RoboDK station: milling.rdk

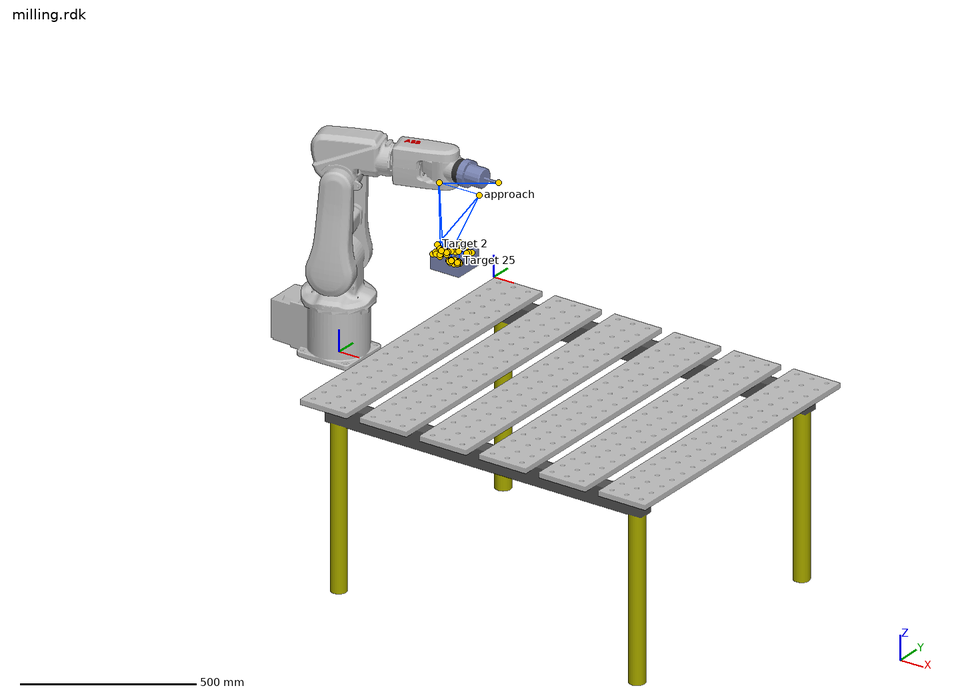
[picture v0: the station drawn from its stored meshes, robots at their saved joint values, targets as dots, program paths as lines]
Station template (saved by RoboDK 5.3.4). Poses are relative to the parent item; angles as X-Y-Z fixed-axis rotations.
  - frame ABB IRB 120-3/0.6 Base at (0, 0, 0) mm
    - robot ABB IRB 120-3/0.6: 6 axes, payload 3 kg, reach 580 mm, repeatability 0.01 mm, weight 25 kg
        modified DH rows (alpha deg, a mm, theta deg, d mm): 0, 0, 0, 290; -90, 0, -90, 0; 0, 270, 0, 0; -90, 70, 0, 302; 90, 0, 0, 0; -90, 0, 180, 72
        joint limits [-165, -110, -90, -160, -120, -400] to [165, 110, 70, 160, 120, 400]; home [0, 0, 0, 0, 0, 0]; saved at [17.579, 3.209, -3.289, -89.746, 17.579, 89.734]
      - tool AssemblyMillCutter, TCP at (0, 0, 112.79) mm, size 80 x 120 x 80 mm
  - object Table at (800, 0, 100) mm, size 1193.8 x 965.2 x 609.6 mm, geometry from welding_table.sld
  - frame worktable at (200, 480, 100) mm
    - object Task3_Part at (250, -430, 280) mm, rotated rx 90 ry 0 rz -180 deg, size 100 x 50 x 100 mm, geometry from Task3_Part.STEP
    - target approach (Cartesian target) at (287, -480, 530) mm, rotated rx 0 ry 90 rz 0 deg; joints [0, 0, 0, 0, 0, 0] of ABB IRB 120-3/0.6
    - target Target 2 (Cartesian target) at (150, -493.7, 340) mm, rotated rx -180 ry 0 rz -90 deg; joints [-2.242, 10.254, -10.083, 0, 89.83, -92.242] of ABB IRB 120-3/0.6
    - target Target 3 (Cartesian target) at (150, -493.7, 320) mm, rotated rx 180 ry 0 rz -90 deg; joints [-2.242, 9.393, -5.327, 0, 85.934, -92.242] of ABB IRB 120-3/0.6
    - target Target 4 (Cartesian target) at (176, -493.7, 320) mm, rotated rx 180 ry 0 rz -90 deg; joints [-2.087, 15.254, -12.292, 0, 87.038, -92.087] of ABB IRB 120-3/0.6
    - target Target 5 (Cartesian target) at (176, -515.9, 320) mm, rotated rx 180 ry 0 rz -90 deg; joints [-5.454, 15.592, -12.71, 0, 87.118, -95.454] of ABB IRB 120-3/0.6
    - target Target 6 (Cartesian target) at (150, -515.9, 320) mm, rotated rx 180 ry 0 rz -90.94 deg; joints [-5.856, 9.74, -5.724, 0, 85.985, -94.918] of ABB IRB 120-3/0.6
    - target Target 7 (Cartesian target) at (150, -501, 320) mm, rotated rx -180 ry 0 rz -90.94 deg; joints [-3.434, 9.473, -5.418, 0, 85.945, -92.496] of ABB IRB 120-3/0.6
    - target Target 8 (Cartesian target) at (170, -501, 320) mm, rotated rx -180 ry 0 rz -90.94 deg; joints [-3.248, 13.955, -10.703, 0, 86.748, -92.31] of ABB IRB 120-3/0.6
    - target Target 9 (Cartesian target) at (157, -508, 320) mm, rotated rx -180 ry 0 rz -90.94 deg; joints [-4.485, 11.132, -7.339, 0, 86.207, -93.547] of ABB IRB 120-3/0.6
    - target Target 10 (Cartesian target) at (170, -508, 320) mm, rotated rx -180 ry 0 rz -90.94 deg; joints [-4.328, 14.06, -10.831, 0, 86.771, -93.39] of ABB IRB 120-3/0.6
    - target Target 11 (Cartesian target) at (170, -508, 340) mm, rotated rx -180 ry 0 rz -90.94 deg; joints [-4.328, 15.03, -15.796, 0, 90.765, -93.39] of ABB IRB 120-3/0.6
    - target Target 24 (Cartesian target) at (194, -444, 340) mm, rotated rx -180 ry 0 rz -90 deg; joints [5.221, 21.03, -23.466, 0, 92.436, -84.779] of ABB IRB 120-3/0.6
    - target Target 13 (Cartesian target) at (194, -444, 320) mm, rotated rx -180 ry 0 rz -90 deg; joints [5.221, 19.845, -18.11, 0, 88.265, -84.779] of ABB IRB 120-3/0.6
    - target Target 14 (Cartesian target) at (236, -444, 320) mm, rotated rx -180 ry 0 rz -90 deg; joints [4.72, 30.95, -33.475, 0, 92.525, -85.28] of ABB IRB 120-3/0.6
    - target Target 15 (Cartesian target) at (236, -466, 320) mm, rotated rx 180 ry 0 rz -90 deg; joints [1.839, 30.578, -32.93, 0, 92.352, -88.161] of ABB IRB 120-3/0.6
    - target Target 16 (Cartesian target) at (194, -466, 320) mm, rotated rx 180 ry 0 rz -90 deg; joints [2.035, 19.507, -17.671, 0, 88.164, -87.965] of ABB IRB 120-3/0.6
    - target Target 17 (Cartesian target) at (194, -450, 320) mm, rotated rx -180 ry 0 rz -90 deg; joints [4.354, 19.724, -17.952, 0, 88.228, -85.646] of ABB IRB 120-3/0.6
    - target Target 18 (Cartesian target) at (229, -450, 320) mm, rotated rx -180 ry 0 rz -90 deg; joints [4, 28.797, -30.354, 0, 91.557, -86] of ABB IRB 120-3/0.6
    - target Target 19 (Cartesian target) at (229, -460, 320) mm, rotated rx -180 ry 0 rz -90 deg; joints [2.669, 28.633, -30.119, 0, 91.486, -87.331] of ABB IRB 120-3/0.6
    - target Target 20 (Cartesian target) at (200, -460, 320) mm, rotated rx -180 ry 0 rz -90 deg; joints [2.862, 21.036, -19.67, 0, 88.635, -87.138] of ABB IRB 120-3/0.6
    - target Target 21 (Cartesian target) at (200, -455, 320) mm, rotated rx -180 ry 0 rz -90 deg; joints [3.576, 21.105, -19.762, 0, 88.657, -86.424] of ABB IRB 120-3/0.6
    - target Target 22 (Cartesian target) at (225, -455, 320) mm, rotated rx -180 ry 0 rz -90 deg; joints [3.366, 27.593, -28.639, 0, 91.046, -86.634] of ABB IRB 120-3/0.6
    - target Target 23 (Cartesian target) at (225, -455, 340) mm, rotated rx -180 ry 0 rz -90 deg; joints [3.366, 29.282, -34.912, 0, 95.63, -86.634] of ABB IRB 120-3/0.6
    - target Target 40 (Cartesian target) at (225, -494, 340) mm, rotated rx -180 ry 0 rz -90 deg; joints [-1.887, 29.131, -34.693, 0, 95.562, -91.887] of ABB IRB 120-3/0.6
    - target Target 25 (Cartesian target) at (225, -494, 310) mm, rotated rx 180 ry 0 rz -90 deg; joints [-1.887, 26.832, -25.67, 0, 88.838, -91.887] of ABB IRB 120-3/0.6
    - target Target 26 (Cartesian target) at (235.62, -501.66, 310) mm, rotated rx -180 ry 0 rz -90 deg; joints [-2.847, 29.827, -29.932, 0, 90.105, -92.847] of ABB IRB 120-3/0.6
    - target Target 27 (Cartesian target) at (225, -516, 310) mm, rotated rx 180 ry 0 rz -90 deg; joints [-4.842, 27.177, -26.154, 0, 88.977, -94.842] of ABB IRB 120-3/0.6
    - target Target 28 (Cartesian target) at (210, -516, 310) mm, rotated rx -180 ry 0 rz -90 deg; joints [-5.018, 23.306, -20.817, 0, 87.511, -95.018] of ABB IRB 120-3/0.6
    - target Target 29 (Cartesian target) at (199.38, -508.34, 310) mm, rotated rx 180 ry 0 rz -90 deg; joints [-4.059, 20.546, -17.146, 0, 86.6, -94.059] of ABB IRB 120-3/0.6
    - target Target 30 (Cartesian target) at (210, -494, 310) mm, rotated rx 180 ry 0 rz -90 deg; joints [-1.956, 22.97, -20.365, 0, 87.394, -91.956] of ABB IRB 120-3/0.6
    - target Target 31 (Cartesian target) at (225, -494, 310) mm, rotated rx -180 ry 0 rz -90 deg; joints [-1.887, 26.832, -25.67, 0, 88.838, -91.887] of ABB IRB 120-3/0.6
    - target Target 32 (Cartesian target) at (232, -501, 310) mm, rotated rx -180 ry 0 rz -90 deg; joints [-2.783, 28.806, -28.465, 0, 89.659, -92.783] of ABB IRB 120-3/0.6
    - target Target 33 (Cartesian target) at (232, -510, 310) mm, rotated rx -180 ry 0 rz -90 deg; joints [-3.972, 28.953, -28.675, 0, 89.722, -93.972] of ABB IRB 120-3/0.6
    - target Target 34 (Cartesian target) at (204, -510, 310) mm, rotated rx -180 ry 0 rz -90 deg; joints [-4.247, 21.7, -18.667, 0, 86.967, -94.247] of ABB IRB 120-3/0.6
    - target Target 35 (Cartesian target) at (204, -500, 310) mm, rotated rx -180 ry 0 rz -90 deg; joints [-2.834, 21.548, -18.466, 0, 86.918, -92.834] of ABB IRB 120-3/0.6
    - target Target 36 (Cartesian target) at (227, -500, 310) mm, rotated rx -180 ry 0 rz -90 deg; joints [-2.682, 27.431, -26.512, 0, 89.081, -92.682] of ABB IRB 120-3/0.6
    - target Target 37 (Cartesian target) at (227, -505, 310) mm, rotated rx -180 ry 0 rz -90 deg; joints [-3.351, 27.502, -26.612, 0, 89.11, -93.351] of ABB IRB 120-3/0.6
    - target Target 38 (Cartesian target) at (207, -505, 310) mm, rotated rx -180 ry 0 rz -90 deg; joints [-3.515, 22.355, -19.54, 0, 87.185, -93.515] of ABB IRB 120-3/0.6
    - target Target 39 (Cartesian target) at (207, -505, 340) mm, rotated rx -180 ry 0 rz -90 deg; joints [-3.515, 24.197, -27.736, 0, 93.539, -93.515] of ABB IRB 120-3/0.6
    - target Target 48 (Cartesian target) at (140, -454, 305) mm, rotated rx -90 ry 0 rz -90 deg; joints [9.51, -28.081, 64.551, 15.739, -37.522, -102.6] of ABB IRB 120-3/0.6
    - target Target 41 (Cartesian target) at (160, -454, 305) mm, rotated rx -90 ry 0 rz -90 deg; joints [8.441, -22.18, 61.05, 13.304, -39.634, -100.321] of ABB IRB 120-3/0.6
    - target Target 42 (Cartesian target) at (160, -462.23, 310.75) mm, rotated rx -90 ry 0 rz -90 deg; joints [5.793, -23.239, 60.543, 9.503, -37.686, -97.546] of ABB IRB 120-3/0.6
    - target Target 43 (Cartesian target) at (160, -466, 305) mm, rotated rx -90 ry 0 rz -90 deg; joints [4.568, -22.569, 61.296, 7.279, -38.953, -95.672] of ABB IRB 120-3/0.6
    - target Target 44 (Cartesian target) at (160, -462.23, 299.55) mm, rotated rx -90 ry 0 rz -90 deg; joints [5.793, -21.695, 61.866, 8.938, -40.516, -96.818] of ABB IRB 120-3/0.6
    - target Target 45 (Cartesian target) at (160, -454, 305) mm, rotated rx -90 ry 0 rz -90 deg; joints [8.441, -22.18, 61.05, 13.304, -39.634, -100.321] of ABB IRB 120-3/0.6
    - target Target 46 (Cartesian target) at (160, -460, 305) mm, rotated rx -90 ry 0 rz -90 deg; joints [6.512, -22.403, 61.191, 10.327, -39.246, -98.032] of ABB IRB 120-3/0.6
    - target Target 47 (Cartesian target) at (140, -460, 305) mm, rotated rx -90 ry 0 rz -90 deg; joints [7.343, -28.357, 64.703, 12.266, -36.98, -99.853] of ABB IRB 120-3/0.6
    - target retract (Cartesian target) at (287, -384.26, 530) mm, rotated rx 0 ry 90 rz 0 deg; joints [17.59, 3.166, -3.244, -89.753, 17.591, 89.741] of ABB IRB 120-3/0.6
    - target Target 49 (Cartesian target) at (147, -480, 530) mm, rotated rx 0 ry 90 rz 0 deg; joints [0, -28.794, 22.363, 0, 6.431, 0] of ABB IRB 120-3/0.6
  - program prog1 (49 instructions, listed below)
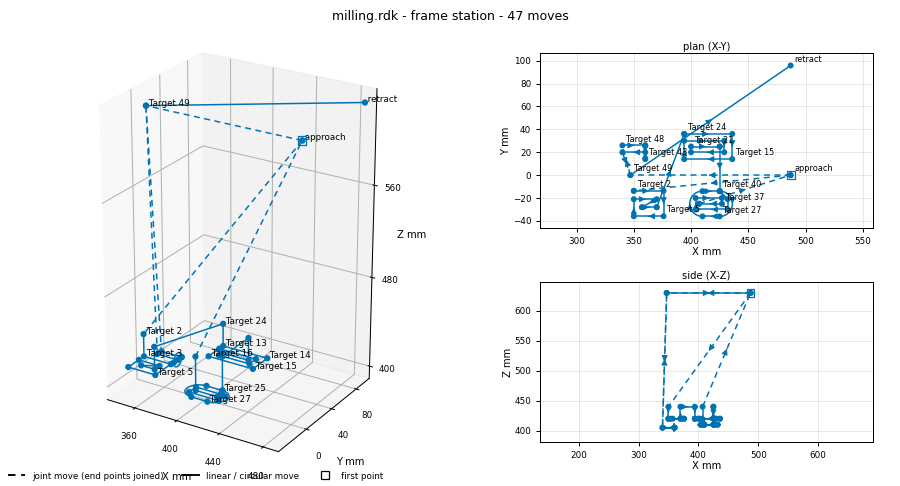
[picture p0: tool path of milling.rdk in frame station, 47 of 47 moves have a stored position in this frame; points joined in program order, loops and branches not executed]

--- program prog1 (robot ABB IRB 120-3/0.6) ---
  设置参考: worktable
  设置工具: AssemblyMillCutter
  MoveJ (approach)
  MoveJ (Target 2)
  MoveL (Target 3)
  MoveL (Target 4)
  MoveL (Target 5)
  MoveL (Target 6)
  MoveL (Target 7)
  MoveL (Target 8)
  MoveL (Target 9)
  MoveL (Target 10)
  MoveL (Target 11)
  MoveL (Target 24)
  MoveL (Target 13)
  MoveL (Target 14)
  MoveL (Target 15)
  MoveL (Target 16)
  MoveL (Target 17)
  MoveL (Target 18)
  MoveL (Target 19)
  MoveL (Target 20)
  MoveL (Target 21)
  MoveL (Target 22)
  MoveL (Target 23)
  MoveL (Target 40)
  MoveL (Target 25)
  MoveC (Target 26, Target 27)
  MoveL (Target 28)
  MoveC (Target 29, Target 30)
  MoveL (Target 31)
  MoveL (Target 32)
  MoveL (Target 33)
  MoveL (Target 34)
  MoveL (Target 35)
  MoveL (Target 36)
  MoveL (Target 37)
  MoveL (Target 38)
  MoveL (Target 39)
  MoveJ (approach)
  MoveJ (Target 49)
  MoveJ (Target 48)
  MoveL (Target 41)
  MoveC (Target 42, Target 43)
  MoveC (Target 44, Target 45)
  MoveL (Target 46)
  MoveL (Target 47)
  MoveJ (Target 49)
  MoveL (retract)
